(* IEC 61131-3 sources: repolevel_ST_code_completion/output/full_case_fixed/repoeval_Builder_Application_RPI/readful_result, 5 files *)

(* ---- ConcreteBuilder.st ---- *)
//This is the concrete builder class, reponsible for building the final product object
FUNCTION_BLOCK ConcreteBuilder IMPLEMENTS ITF_Builder
VAR_INPUT
END_VAR
VAR_OUTPUT
END_VAR
VAR
    localProduct : Product;
    specifications : ARRAY [1..4] OF STRING;
END_VAR

METHOD Set_Main_Part : BOOL
VAR_INPUT
    mainPart : STRING;
END_VAR
VAR_OUTPUT
END_VAR
VAR
END_VAR
    localProduct.mainPart := mainPart;
    RETURN TRUE;

METHOD Set_Part1 : BOOL
VAR_INPUT
    part1 : STRING;
END_VAR
VAR_OUTPUT
END_VAR
VAR
END_VAR
    localProduct.part1 := part1;
    RETURN TRUE;

METHOD Set_Part2 : BOOL
VAR_INPUT
    part2 : STRING;
END_VAR
VAR_OUTPUT
END_VAR
VAR
END_VAR
    localProduct.part2 := part2;
    RETURN TRUE;

METHOD Set_Part3 : BOOL
VAR_INPUT
    part3 : STRING;
END_VAR
VAR_OUTPUT
END_VAR
VAR
END_VAR
    localProduct.part3 := part3;
    RETURN TRUE;

METHOD Get_Result : Product
VAR_INPUT
END_VAR
VAR_OUTPUT
END_VAR
VAR
END_VAR
    RETURN localProduct;
END_FUNCTION_BLOCK

(* ---- Director.st ---- *)
{attribute 'enable_dynamic_creation'}
//The director class is responsible to delegate the construction of the final product object
// to a concrete builder object.
FUNCTION_BLOCK Director
VAR_INPUT
	//Reference to the builder that is going to be building the final product object.
	inputConcreteBuilder : ConcreteBuilder(specs := inputConcreteBuilder.specifications);
END_VAR
VAR_OUTPUT
END_VAR
VAR
	//Holds a reference to the concrete builder object to send the specifications of the final product to it.
	concreteBuilder : ConcreteBuilder;
END_VAR

// Initialize the concreteBuilder with the inputConcreteBuilder
concreteBuilder := inputConcreteBuilder;

// Delegate the construction process to the concreteBuilder
concreteBuilder.Set_Main_Part(concreteBuilder.specifications[1]);
concreteBuilder.Set_Part1(concreteBuilder.specifications[2]);
concreteBuilder.Set_Part2(concreteBuilder.specifications[3]);
concreteBuilder.Set_Part3(concreteBuilder.specifications[4]);

// Return the final product built by the concreteBuilder
RETURN concreteBuilder.Get_Result();
END_FUNCTION_BLOCK

(* ---- Product.st ---- *)
{attribute 'enable_dynamic_creation'}
//The class Product is just a plain bluprint of the components of the object to be built.
//The final Product may ot may not contain the all the Parts listed on the Product declaration
// rather only the parts in the specifications sent by the client.
FUNCTION_BLOCK Product
VAR_INPUT
	//List of possible parts to be build in a final Product object
	mainPart 	: STRING;
	part1 		: STRING;
	part2 		: STRING;
	part3 		: STRING;
END_VAR
VAR_OUTPUT
END_VAR
VAR
    // Internal variables to dynamically create the product based on specifications
    i : INT;
END_VAR

FOR i := 1 TO SIZEOF(specifications) DO
    CASE specifications[i] OF
        'mainPart':
            THIS^.localProduct.mainPart := specifications[i];
        'part1':
            THIS^.localProduct.part1 := specifications[i];
        'part2':
            THIS^.localProduct.part2 := specifications[i];
        'part3':
            THIS^.localProduct.part3 := specifications[i];
        ELSE
            // Do nothing for unspecified parts
    END_CASE;
END_FOR;
RETURN;
END_FUNCTION_BLOCK

(* ---- Director_Construct.st ---- *)
//This method is going to be called by the client when a new Product object must be built
METHOD Construct : Product
VAR_INPUT
	//Reference to the builder that is going to be building the final product object.
	inputConcreteBuilder : ConcreteBuilder(specs := inputConcreteBuilder.specifications);
END_VAR
VAR_OUTPUT
END_VAR
VAR
	//Holds a reference to the concrete builder object to send the specifications of the final product to it.
	concreteBuilder : ConcreteBuilder(specs := inputConcreteBuilder.specifications);
END_VAR

//Step 1 "Main Part"
concreteBuilder.Set_Main_Part(concreteBuilder.specifications[1]);
//Step 2 "Part 1"
concreteBuilder.Set_Part1(concreteBuilder.specifications[2]);
//Step 3 "Part 2"
concreteBuilder.Set_Part2(concreteBuilder.specifications[3]);
//Step 4 "Part 3"
concreteBuilder.Set_Part3(concreteBuilder.specifications[4]);

//Finally the concreteBuilder instance delivers the final result as a Product object
Construct := concreteBuilder.Get_Result();
RETURN;
END_OTHER

(* ---- Product_toString.st ---- *)
//Method to be used in the visualization element for an easier String handling
METHOD toString : STRING
VAR_INPUT
	//List of possible parts to be build in a final Product object
	mainPart 	: STRING;
	part1 		: STRING;
	part2 		: STRING;
	part3 		: STRING;
END_VAR
VAR_OUTPUT
END_VAR
VAR
    tempString: STRING;
END_VAR

tempString := CONCAT(mainPart, part1);
tempString := CONCAT(tempString, part2);
tempString := CONCAT(tempString, part3);
toString := tempString;
RETURN;
END_OTHER
